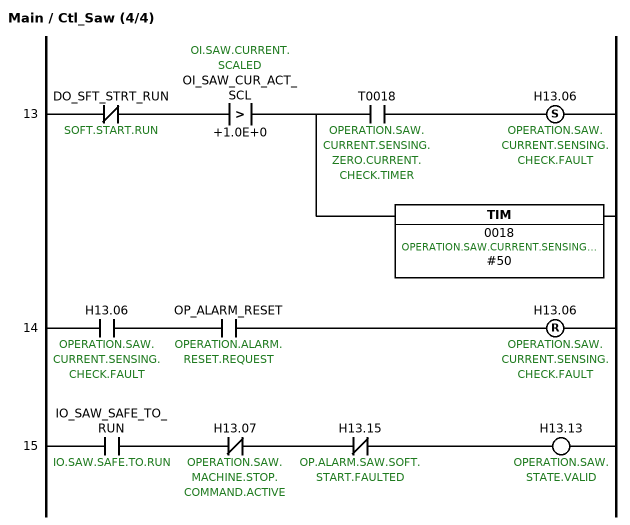
; [picture p72: Main / Ctl_Saw, rungs 13-15]
; rung 13
LDNOT DO_SFT_STRT_RUN  ; SOFT.START.RUN
AND>F(333) OI_SAW_CUR_ACT_SCL +1.0E+0  ; OI.SAW.CURRENT.SCALED
OUT TR0
AND T0018  ; OPERATION.SAW.CURRENT.SENSING.ZERO.CURRENT.CHECK.TIMER
SET H13.06  ; OPERATION.SAW.CURRENT.SENSING.CHECK.FAULT
LD TR0
TIM 0018 #50  ; OPERATION.SAW.CURRENT.SENSING.ZERO.CURRENT.CHECK.TIMER
; rung 14
LD H13.06  ; OPERATION.SAW.CURRENT.SENSING.CHECK.FAULT
AND OP_ALARM_RESET  ; OPERATION.ALARM.RESET.REQUEST
RSET H13.06  ; OPERATION.SAW.CURRENT.SENSING.CHECK.FAULT
; rung 15
LD IO_SAW_SAFE_TO_RUN  ; IO.SAW.SAFE.TO.RUN
ANDNOT H13.07  ; OPERATION.SAW.MACHINE.STOP.COMMAND.ACTIVE
ANDNOT H13.15  ; OP.ALARM.SAW.SOFT.START.FAULTED
OUT H13.13  ; OPERATION.SAW.STATE.VALID

### Section Ctl_Water

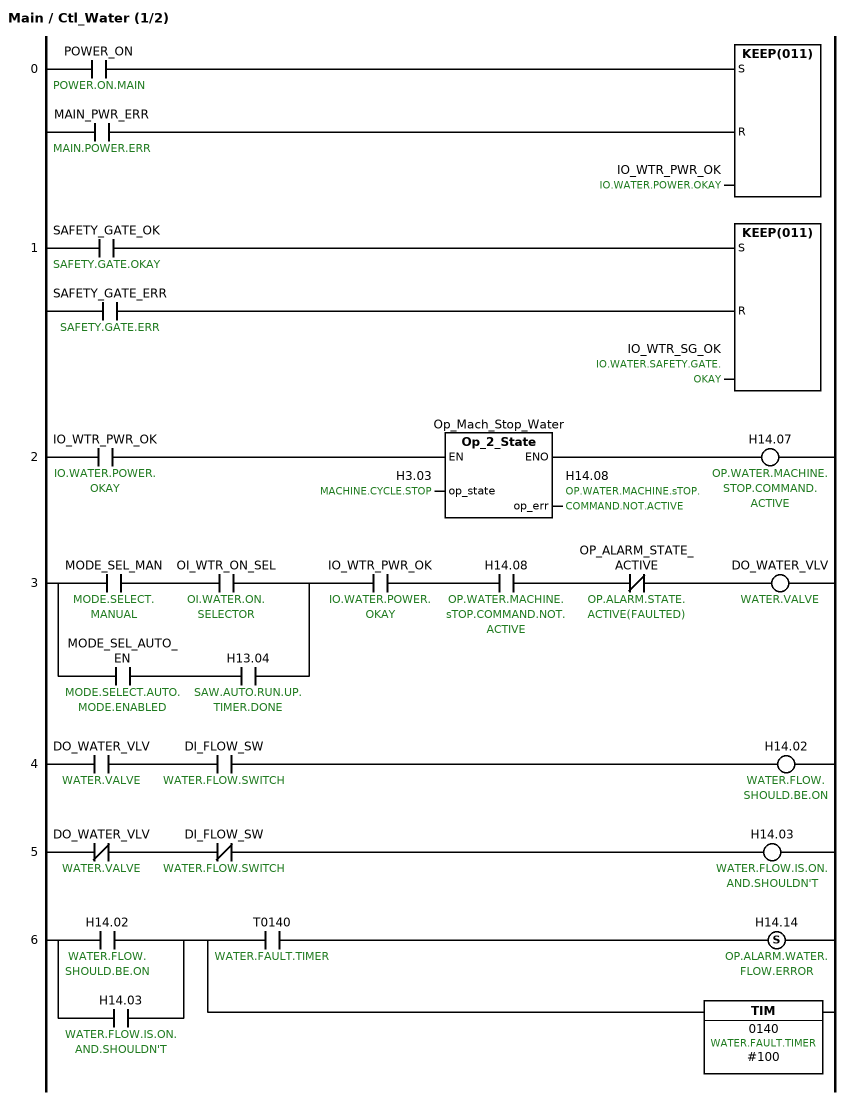
; rung 0
LD POWER_ON  ; POWER.ON.MAIN
LD MAIN_PWR_ERR  ; MAIN.POWER.ERR
KEEP(011) IO_WTR_PWR_OK  ; IO.WATER.POWER.OKAY
; rung 1
LD SAFETY_GATE_OK  ; SAFETY.GATE.OKAY
LD SAFETY_GATE_ERR  ; SAFETY.GATE.ERR
KEEP(011) IO_WTR_SG_OK  ; IO.WATER.SAFETY.GATE.OKAY
; rung 2
LD IO_WTR_PWR_OK  ; IO.WATER.POWER.OKAY
CALL Op_Mach_Stop_Water : Op_2_State (op_state := H3.03, op_err => H14.08)  ; MACHINE.CYCLE.STOP, OP.WATER.MACHINE.sTOP.COMMAND.NOT.ACTIVE
OUT H14.07  ; OP.WATER.MACHINE.STOP.COMMAND.ACTIVE
; rung 3
LD MODE_SEL_MAN  ; MODE.SELECT.MANUAL
AND OI_WTR_ON_SEL  ; OI.WATER.ON.SELECTOR
LD MODE_SEL_AUTO_EN  ; MODE.SELECT.AUTO.MODE.ENABLED
AND H13.04  ; SAW.AUTO.RUN.UP.TIMER.DONE
ORLD
AND IO_WTR_PWR_OK  ; IO.WATER.POWER.OKAY
AND H14.08  ; OP.WATER.MACHINE.sTOP.COMMAND.NOT.ACTIVE
ANDNOT OP_ALARM_STATE_ACTIVE  ; OP.ALARM.STATE.ACTIVE(FAULTED)
OUT DO_WATER_VLV  ; WATER.VALVE
; rung 4
LD DO_WATER_VLV  ; WATER.VALVE
AND DI_FLOW_SW  ; WATER.FLOW.SWITCH
OUT H14.02  ; WATER.FLOW.SHOULD.BE.ON
; rung 5
LDNOT DO_WATER_VLV  ; WATER.VALVE
ANDNOT DI_FLOW_SW  ; WATER.FLOW.SWITCH
OUT H14.03  ; WATER.FLOW.IS.ON.AND.SHOULDN'T
; rung 6
LD H14.02  ; WATER.FLOW.SHOULD.BE.ON
OR H14.03  ; WATER.FLOW.IS.ON.AND.SHOULDN'T
OUT TR0
AND T0140  ; WATER.FAULT.TIMER
SET H14.14  ; OP.ALARM.WATER.FLOW.ERROR
LD TR0
TIM 0140 #100  ; WATER.FAULT.TIMER

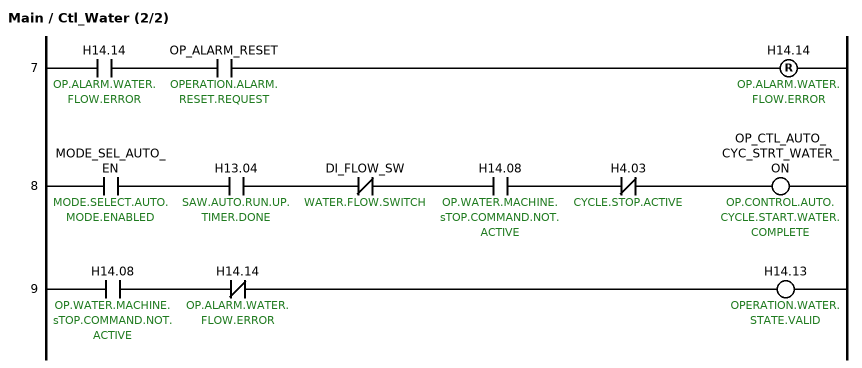
; rung 7
LD H14.14  ; OP.ALARM.WATER.FLOW.ERROR
AND OP_ALARM_RESET  ; OPERATION.ALARM.RESET.REQUEST
RSET H14.14  ; OP.ALARM.WATER.FLOW.ERROR
; rung 8
LD MODE_SEL_AUTO_EN  ; MODE.SELECT.AUTO.MODE.ENABLED
AND H13.04  ; SAW.AUTO.RUN.UP.TIMER.DONE
ANDNOT DI_FLOW_SW  ; WATER.FLOW.SWITCH
AND H14.08  ; OP.WATER.MACHINE.sTOP.COMMAND.NOT.ACTIVE
ANDNOT H4.03  ; CYCLE.STOP.ACTIVE
OUT OP_CTL_AUTO_CYC_STRT_WATER_ON  ; OP.CONTROL.AUTO.CYCLE.START.WATER.COMPLETE
; rung 9
LD H14.08  ; OP.WATER.MACHINE.sTOP.COMMAND.NOT.ACTIVE
ANDNOT H14.14  ; OP.ALARM.WATER.FLOW.ERROR
OUT H14.13  ; OPERATION.WATER.STATE.VALID

### Section Ctl_Lazer

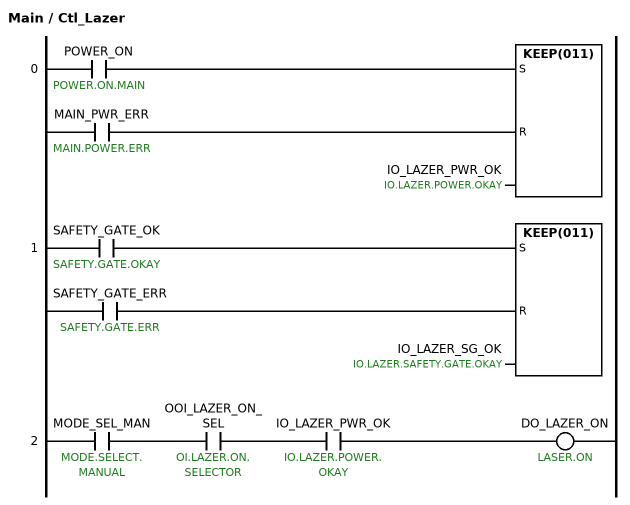
; rung 0
LD POWER_ON  ; POWER.ON.MAIN
LD MAIN_PWR_ERR  ; MAIN.POWER.ERR
KEEP(011) IO_LAZER_PWR_OK  ; IO.LAZER.POWER.OKAY
; rung 1
LD SAFETY_GATE_OK  ; SAFETY.GATE.OKAY
LD SAFETY_GATE_ERR  ; SAFETY.GATE.ERR
KEEP(011) IO_LAZER_SG_OK  ; IO.LAZER.SAFETY.GATE.OKAY
; rung 2
LD MODE_SEL_MAN  ; MODE.SELECT.MANUAL
AND OOI_LAZER_ON_SEL  ; OI.LAZER.ON.SELECTOR
AND IO_LAZER_PWR_OK  ; IO.LAZER.POWER.OKAY
OUT DO_LAZER_ON  ; LASER.ON

### Section Init_Recipe

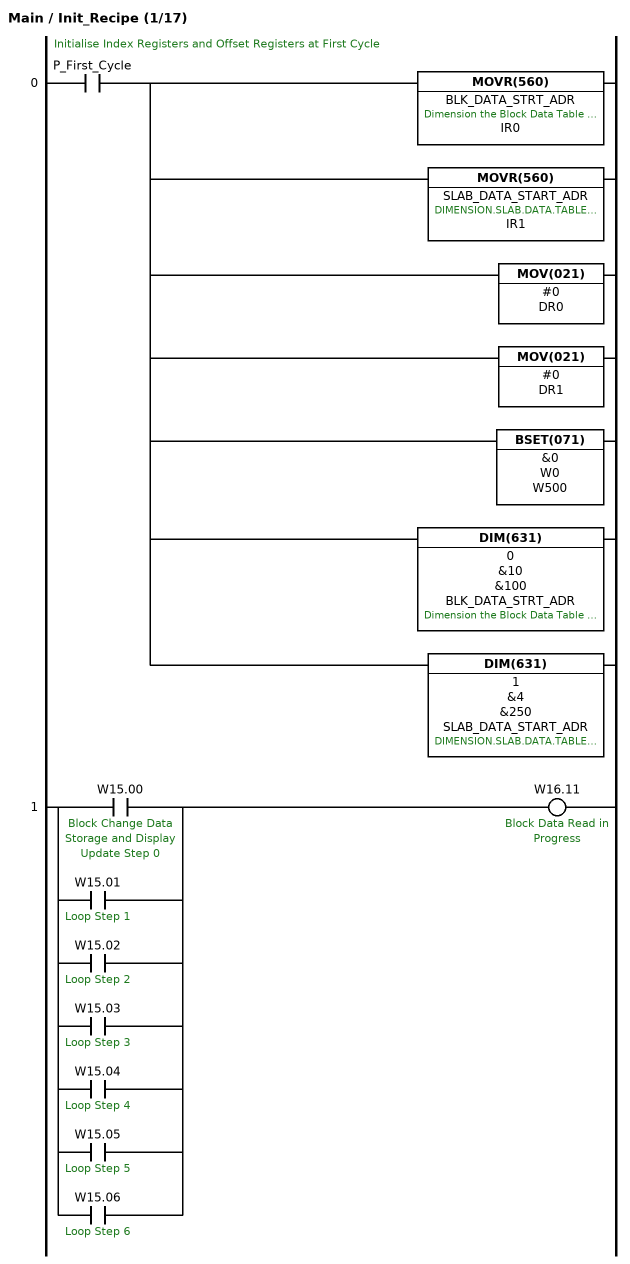
; rung 0: Initialise Index Registers and Offset Registers at First Cycle
LD P_First_Cycle
MOVR(560) BLK_DATA_STRT_ADR IR0  ; Dimension the Block Data Table - Start Address
MOVR(560) SLAB_DATA_START_ADR IR1  ; DIMENSION.SLAB.DATA.TABLE.START.ADDRESS
MOV(021) #0 DR0
MOV(021) #0 DR1
BSET(071) &0 W0 W500
DIM(631) 0 &10 &100 BLK_DATA_STRT_ADR  ; Dimension the Block Data Table - Start Address
DIM(631) 1 &4 &250 SLAB_DATA_START_ADR  ; DIMENSION.SLAB.DATA.TABLE.START.ADDRESS
; rung 1
LD W15.00  ; Block Change Data Storage and Display Update Step 0
OR W15.01  ; Loop Step 1
OR W15.02  ; Loop Step 2
OR W15.03  ; Loop Step 3
OR W15.04  ; Loop Step 4
OR W15.05  ; Loop Step 5
OR W15.06  ; Loop Step 6
OUT W16.11  ; Block Data Read in Progress

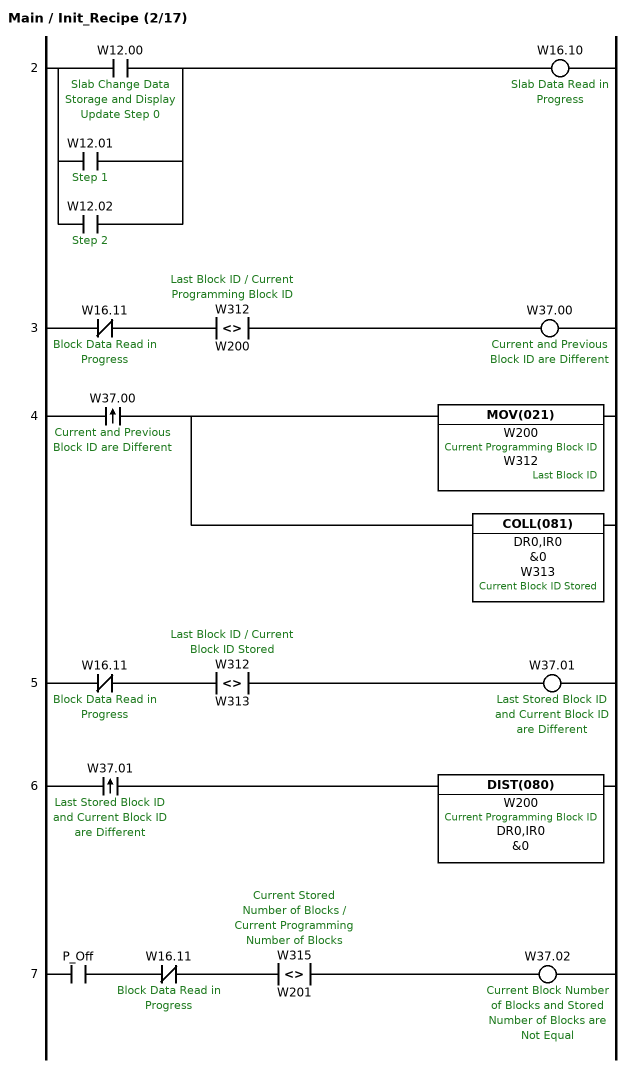
; rung 2
LD W12.00  ; Slab Change Data Storage and Display Update Step 0
OR W12.01  ; Step 1
OR W12.02  ; Step 2
OUT W16.10  ; Slab Data Read in Progress
; rung 3
LDNOT W16.11  ; Block Data Read in Progress
AND<>(305) W312 W200  ; Last Block ID, Current Programming Block ID
OUT W37.00  ; Current and Previous Block ID are Different
; rung 4
@LD W37.00  ; Current and Previous Block ID are Different
MOV(021) W200 W312  ; Current Programming Block ID, Last Block ID
COLL(081) DR0,IR0 &0 W313  ; Current Block ID Stored
; rung 5
LDNOT W16.11  ; Block Data Read in Progress
AND<>(305) W312 W313  ; Last Block ID, Current Block ID Stored
OUT W37.01  ; Last Stored Block ID and Current Block ID are Different
; rung 6
@LD W37.01  ; Last Stored Block ID and Current Block ID are Different
DIST(080) W200 DR0,IR0 &0  ; Current Programming Block ID
; rung 7
LD P_Off
ANDNOT W16.11  ; Block Data Read in Progress
AND<>(305) W315 W201  ; Current Stored Number of Blocks, Current Programming Number of Blocks
OUT W37.02  ; Current Block Number of Blocks and Stored Number of Blocks are Not Equal

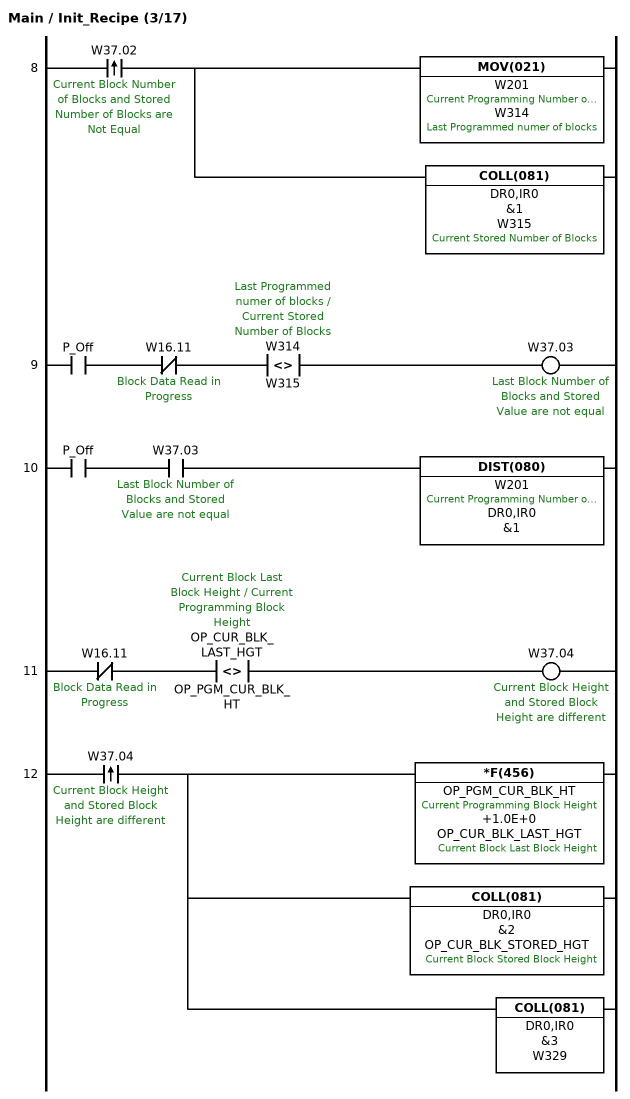
; rung 8
@LD W37.02  ; Current Block Number of Blocks and Stored Number of Blocks are Not Equal
MOV(021) W201 W314  ; Current Programming Number of Blocks, Last Programmed numer of blocks
COLL(081) DR0,IR0 &1 W315  ; Current Stored Number of Blocks
; rung 9
LD P_Off
ANDNOT W16.11  ; Block Data Read in Progress
AND<>(305) W314 W315  ; Last Programmed numer of blocks, Current Stored Number of Blocks
OUT W37.03  ; Last Block Number of Blocks and Stored Value are not equal
; rung 10
LD P_Off
AND W37.03  ; Last Block Number of Blocks and Stored Value are not equal
DIST(080) W201 DR0,IR0 &1  ; Current Programming Number of Blocks
; rung 11
LDNOT W16.11  ; Block Data Read in Progress
AND<>F(330) OP_CUR_BLK_LAST_HGT OP_PGM_CUR_BLK_HT  ; Current Block Last Block Height, Current Programming Block Height
OUT W37.04  ; Current Block Height and Stored Block Height are different
; rung 12
@LD W37.04  ; Current Block Height and Stored Block Height are different
*F(456) OP_PGM_CUR_BLK_HT +1.0E+0 OP_CUR_BLK_LAST_HGT  ; Current Programming Block Height, Current Block Last Block Height
COLL(081) DR0,IR0 &2 OP_CUR_BLK_STORED_HGT  ; Current Block Stored Block Height
COLL(081) DR0,IR0 &3 W329

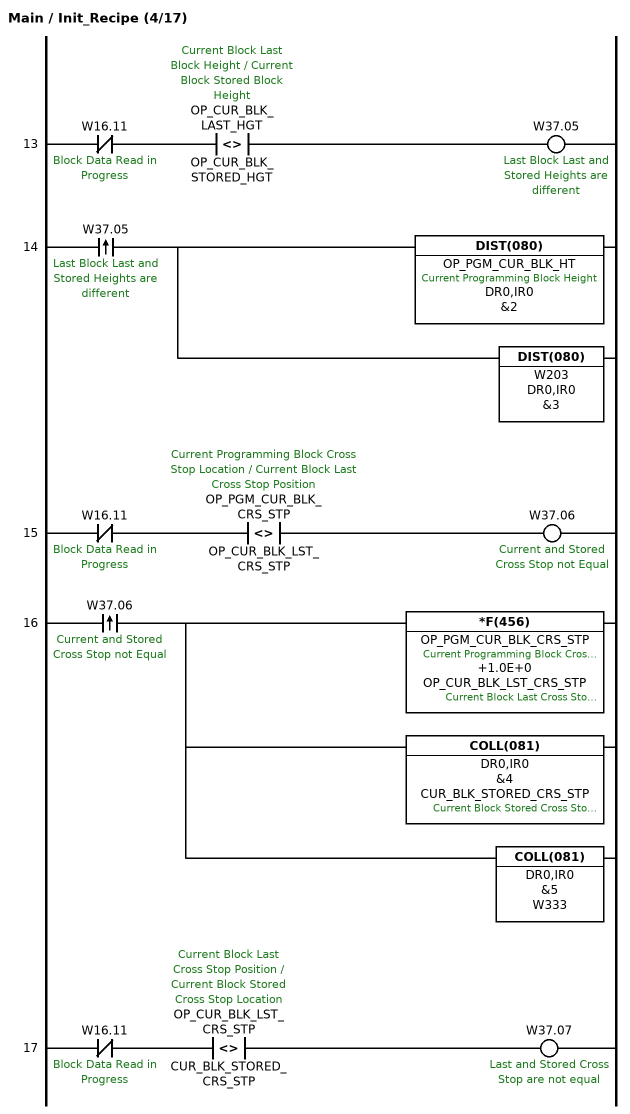
; rung 13
LDNOT W16.11  ; Block Data Read in Progress
AND<>F(330) OP_CUR_BLK_LAST_HGT OP_CUR_BLK_STORED_HGT  ; Current Block Last Block Height, Current Block Stored Block Height
OUT W37.05  ; Last Block Last and Stored Heights are different
; rung 14
@LD W37.05  ; Last Block Last and Stored Heights are different
DIST(080) OP_PGM_CUR_BLK_HT DR0,IR0 &2  ; Current Programming Block Height
DIST(080) W203 DR0,IR0 &3
; rung 15
LDNOT W16.11  ; Block Data Read in Progress
AND<>F(330) OP_PGM_CUR_BLK_CRS_STP OP_CUR_BLK_LST_CRS_STP  ; Current Programming Block Cross Stop Location, Current Block Last Cross Stop Position
OUT W37.06  ; Current and Stored Cross Stop not Equal
; rung 16
@LD W37.06  ; Current and Stored Cross Stop not Equal
*F(456) OP_PGM_CUR_BLK_CRS_STP +1.0E+0 OP_CUR_BLK_LST_CRS_STP  ; Current Programming Block Cross Stop Location, Current Block Last Cross Stop Position
COLL(081) DR0,IR0 &4 CUR_BLK_STORED_CRS_STP  ; Current Block Stored Cross Stop Location
COLL(081) DR0,IR0 &5 W333
; rung 17
LDNOT W16.11  ; Block Data Read in Progress
AND<>F(330) OP_CUR_BLK_LST_CRS_STP CUR_BLK_STORED_CRS_STP  ; Current Block Last Cross Stop Position, Current Block Stored Cross Stop Location
OUT W37.07  ; Last and Stored Cross Stop are not equal

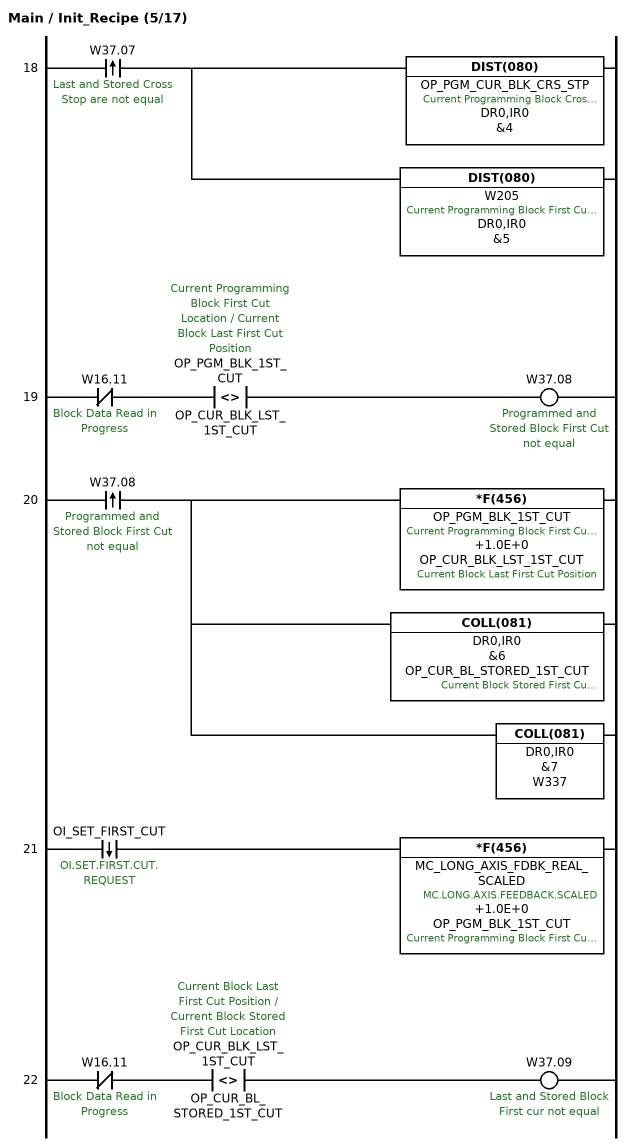
; rung 18
@LD W37.07  ; Last and Stored Cross Stop are not equal
DIST(080) OP_PGM_CUR_BLK_CRS_STP DR0,IR0 &4  ; Current Programming Block Cross Stop Location
DIST(080) W205 DR0,IR0 &5  ; Current Programming Block First Cut Location
; rung 19
LDNOT W16.11  ; Block Data Read in Progress
AND<>F(330) OP_PGM_BLK_1ST_CUT OP_CUR_BLK_LST_1ST_CUT  ; Current Programming Block First Cut Location, Current Block Last First Cut Position
OUT W37.08  ; Programmed and Stored Block First Cut not equal
; rung 20
@LD W37.08  ; Programmed and Stored Block First Cut not equal
*F(456) OP_PGM_BLK_1ST_CUT +1.0E+0 OP_CUR_BLK_LST_1ST_CUT  ; Current Programming Block First Cut Location, Current Block Last First Cut Position
COLL(081) DR0,IR0 &6 OP_CUR_BL_STORED_1ST_CUT  ; Current Block Stored First Cut Location
COLL(081) DR0,IR0 &7 W337
; rung 21
%LD OI_SET_FIRST_CUT  ; OI.SET.FIRST.CUT.REQUEST
*F(456) MC_LONG_AXIS_FDBK_REAL_SCALED +1.0E+0 OP_PGM_BLK_1ST_CUT  ; MC.LONG.AXIS.FEEDBACK.SCALED, Current Programming Block First Cut Location
; rung 22
LDNOT W16.11  ; Block Data Read in Progress
AND<>F(330) OP_CUR_BLK_LST_1ST_CUT OP_CUR_BL_STORED_1ST_CUT  ; Current Block Last First Cut Position, Current Block Stored First Cut Location
OUT W37.09  ; Last and Stored Block First cur not equal

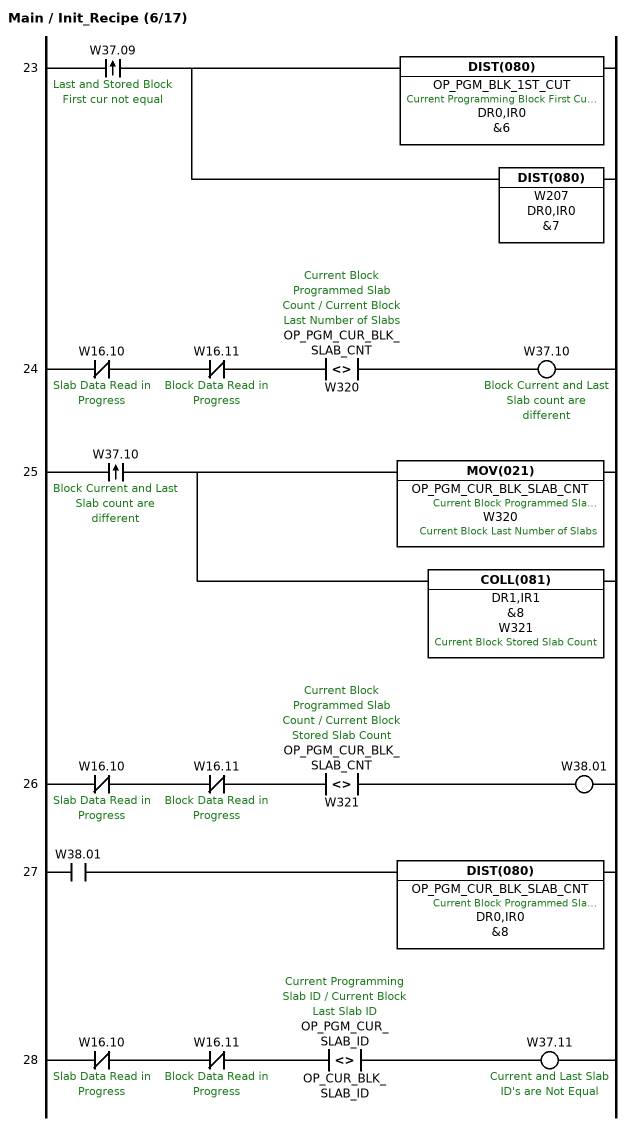
; rung 23
@LD W37.09  ; Last and Stored Block First cur not equal
DIST(080) OP_PGM_BLK_1ST_CUT DR0,IR0 &6  ; Current Programming Block First Cut Location
DIST(080) W207 DR0,IR0 &7
; rung 24
LDNOT W16.10  ; Slab Data Read in Progress
ANDNOT W16.11  ; Block Data Read in Progress
AND<>(305) OP_PGM_CUR_BLK_SLAB_CNT W320  ; Current Block Programmed Slab Count, Current Block Last Number of Slabs
OUT W37.10  ; Block Current and Last Slab count are different
; rung 25
@LD W37.10  ; Block Current and Last Slab count are different
MOV(021) OP_PGM_CUR_BLK_SLAB_CNT W320  ; Current Block Programmed Slab Count, Current Block Last Number of Slabs
COLL(081) DR1,IR1 &8 W321  ; Current Block Stored Slab Count
; rung 26
LDNOT W16.10  ; Slab Data Read in Progress
ANDNOT W16.11  ; Block Data Read in Progress
AND<>(305) OP_PGM_CUR_BLK_SLAB_CNT W321  ; Current Block Programmed Slab Count, Current Block Stored Slab Count
OUT W38.01
; rung 27
LD W38.01
DIST(080) OP_PGM_CUR_BLK_SLAB_CNT DR0,IR0 &8  ; Current Block Programmed Slab Count
; rung 28
LDNOT W16.10  ; Slab Data Read in Progress
ANDNOT W16.11  ; Block Data Read in Progress
AND<>(305) OP_PGM_CUR_SLAB_ID OP_CUR_BLK_SLAB_ID  ; Current Programming Slab ID, Current Block Last Slab ID
OUT W37.11  ; Current and Last Slab ID's are Not Equal

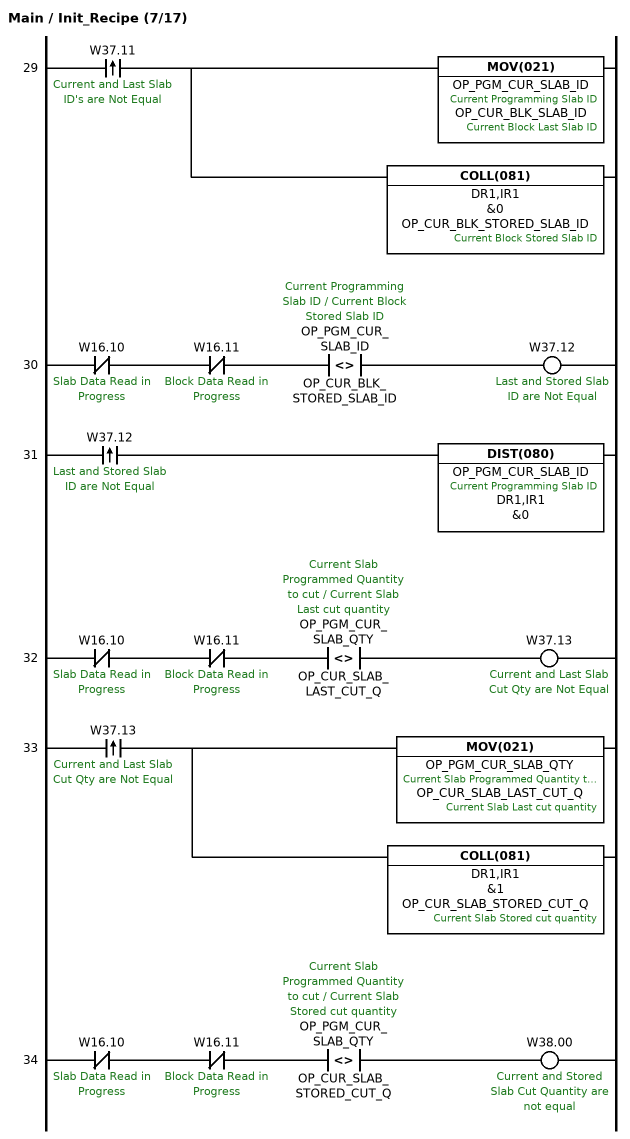
; rung 29
@LD W37.11  ; Current and Last Slab ID's are Not Equal
MOV(021) OP_PGM_CUR_SLAB_ID OP_CUR_BLK_SLAB_ID  ; Current Programming Slab ID, Current Block Last Slab ID
COLL(081) DR1,IR1 &0 OP_CUR_BLK_STORED_SLAB_ID  ; Current Block Stored Slab ID
; rung 30
LDNOT W16.10  ; Slab Data Read in Progress
ANDNOT W16.11  ; Block Data Read in Progress
AND<>(305) OP_PGM_CUR_SLAB_ID OP_CUR_BLK_STORED_SLAB_ID  ; Current Programming Slab ID, Current Block Stored Slab ID
OUT W37.12  ; Last and Stored Slab ID are Not Equal
; rung 31
@LD W37.12  ; Last and Stored Slab ID are Not Equal
DIST(080) OP_PGM_CUR_SLAB_ID DR1,IR1 &0  ; Current Programming Slab ID
; rung 32
LDNOT W16.10  ; Slab Data Read in Progress
ANDNOT W16.11  ; Block Data Read in Progress
AND<>(305) OP_PGM_CUR_SLAB_QTY OP_CUR_SLAB_LAST_CUT_Q  ; Current Slab Programmed Quantity to cut, Current Slab Last cut quantity
OUT W37.13  ; Current and Last Slab Cut Qty are Not Equal
; rung 33
@LD W37.13  ; Current and Last Slab Cut Qty are Not Equal
MOV(021) OP_PGM_CUR_SLAB_QTY OP_CUR_SLAB_LAST_CUT_Q  ; Current Slab Programmed Quantity to cut, Current Slab Last cut quantity
COLL(081) DR1,IR1 &1 OP_CUR_SLAB_STORED_CUT_Q  ; Current Slab Stored cut quantity
; rung 34
LDNOT W16.10  ; Slab Data Read in Progress
ANDNOT W16.11  ; Block Data Read in Progress
AND<>(305) OP_PGM_CUR_SLAB_QTY OP_CUR_SLAB_STORED_CUT_Q  ; Current Slab Programmed Quantity to cut, Current Slab Stored cut quantity
OUT W38.00  ; Current and Stored Slab Cut Quantity are not equal

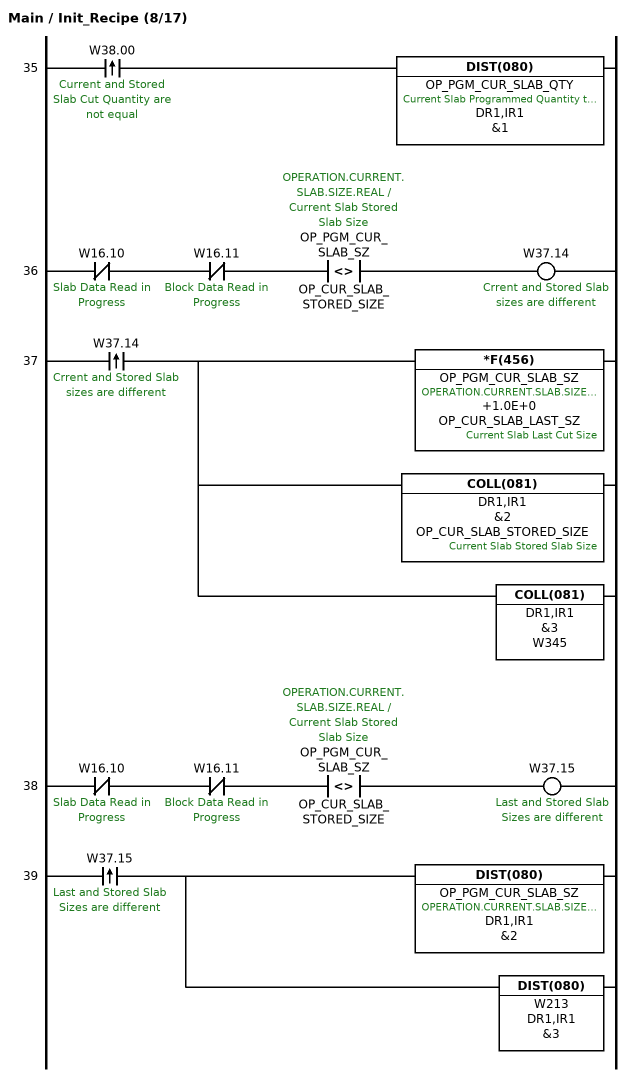
; rung 35
@LD W38.00  ; Current and Stored Slab Cut Quantity are not equal
DIST(080) OP_PGM_CUR_SLAB_QTY DR1,IR1 &1  ; Current Slab Programmed Quantity to cut
; rung 36
LDNOT W16.10  ; Slab Data Read in Progress
ANDNOT W16.11  ; Block Data Read in Progress
AND<>F(330) OP_PGM_CUR_SLAB_SZ OP_CUR_SLAB_STORED_SIZE  ; OPERATION.CURRENT.SLAB.SIZE.REAL, Current Slab Stored Slab Size
OUT W37.14  ; Crrent and Stored Slab sizes are different
; rung 37
@LD W37.14  ; Crrent and Stored Slab sizes are different
*F(456) OP_PGM_CUR_SLAB_SZ +1.0E+0 OP_CUR_SLAB_LAST_SZ  ; OPERATION.CURRENT.SLAB.SIZE.REAL, Current Slab Last Cut Size
COLL(081) DR1,IR1 &2 OP_CUR_SLAB_STORED_SIZE  ; Current Slab Stored Slab Size
COLL(081) DR1,IR1 &3 W345
; rung 38
LDNOT W16.10  ; Slab Data Read in Progress
ANDNOT W16.11  ; Block Data Read in Progress
AND<>F(330) OP_PGM_CUR_SLAB_SZ OP_CUR_SLAB_STORED_SIZE  ; OPERATION.CURRENT.SLAB.SIZE.REAL, Current Slab Stored Slab Size
OUT W37.15  ; Last and Stored Slab Sizes are different
; rung 39
@LD W37.15  ; Last and Stored Slab Sizes are different
DIST(080) OP_PGM_CUR_SLAB_SZ DR1,IR1 &2  ; OPERATION.CURRENT.SLAB.SIZE.REAL
DIST(080) W213 DR1,IR1 &3

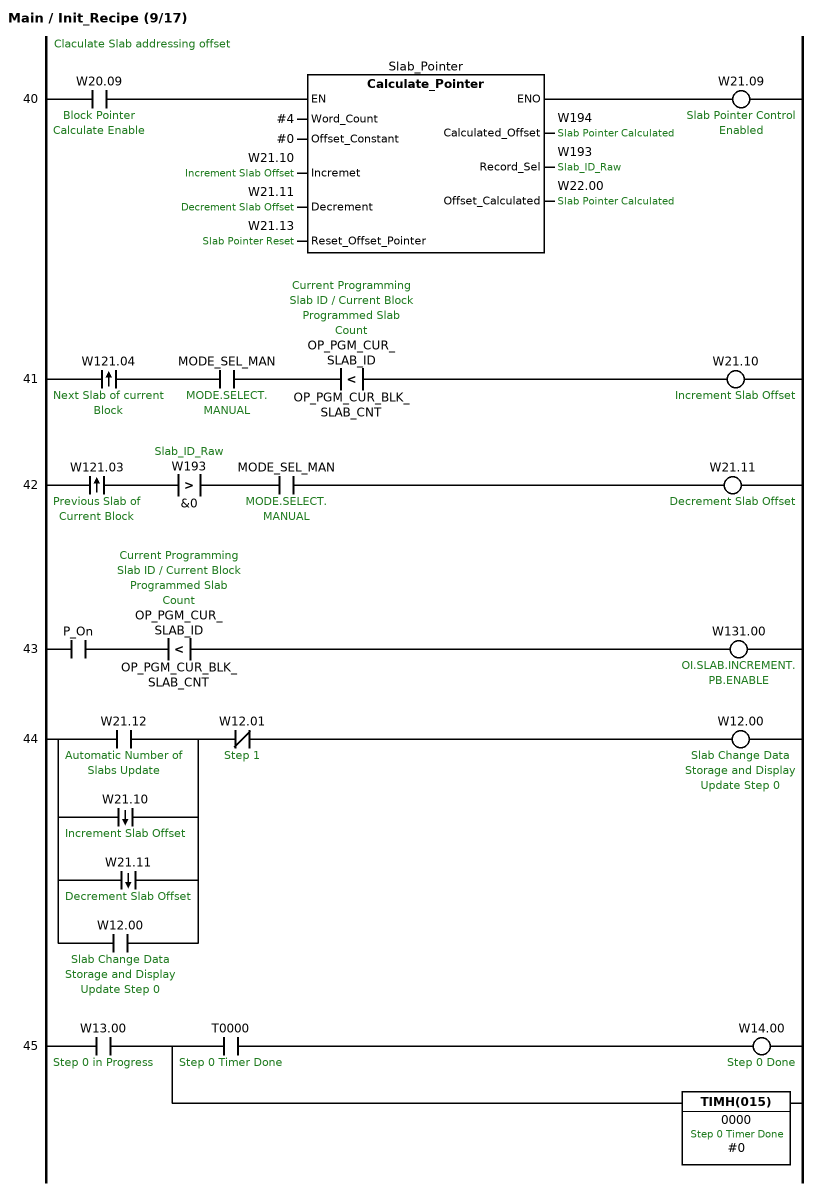
; rung 40: Claculate Slab addressing offset
LD W20.09  ; Block Pointer Calculate Enable
CALL Slab_Pointer : Calculate_Pointer (Word_Count := #4, Offset_Constant := #0, Incremet := W21.10, Decrement := W21.11, Reset_Offset_Pointer := W21.13, Calculated_Offset => W194, Record_Sel => W193, Offset_Calculated => W22.00)  ; Increment Slab Offset, Decrement Slab Offset, Slab Pointer Reset, Slab Pointer Calculated, Slab_ID_Raw
OUT W21.09  ; Slab Pointer Control Enabled
; rung 41
@LD W121.04  ; Next Slab of current Block
AND MODE_SEL_MAN  ; MODE.SELECT.MANUAL
AND<(310) OP_PGM_CUR_SLAB_ID OP_PGM_CUR_BLK_SLAB_CNT  ; Current Programming Slab ID, Current Block Programmed Slab Count
OUT W21.10  ; Increment Slab Offset
; rung 42
@LD W121.03  ; Previous Slab of Current Block
AND>(320) W193 &0  ; Slab_ID_Raw
AND MODE_SEL_MAN  ; MODE.SELECT.MANUAL
OUT W21.11  ; Decrement Slab Offset
; rung 43
LD P_On
AND<(310) OP_PGM_CUR_SLAB_ID OP_PGM_CUR_BLK_SLAB_CNT  ; Current Programming Slab ID, Current Block Programmed Slab Count
OUT W131.00  ; OI.SLAB.INCREMENT.PB.ENABLE
; rung 44
LD W21.12  ; Automatic Number of Slabs Update
%OR W21.10  ; Increment Slab Offset
%OR W21.11  ; Decrement Slab Offset
OR W12.00  ; Slab Change Data Storage and Display Update Step 0
ANDNOT W12.01  ; Step 1
OUT W12.00  ; Slab Change Data Storage and Display Update Step 0
; rung 45
LD W13.00  ; Step 0 in Progress
OUT TR0
AND T0000  ; Step 0 Timer Done
OUT W14.00  ; Step 0 Done
LD TR0
TIMH(015) 0000 #0  ; Step 0 Timer Done

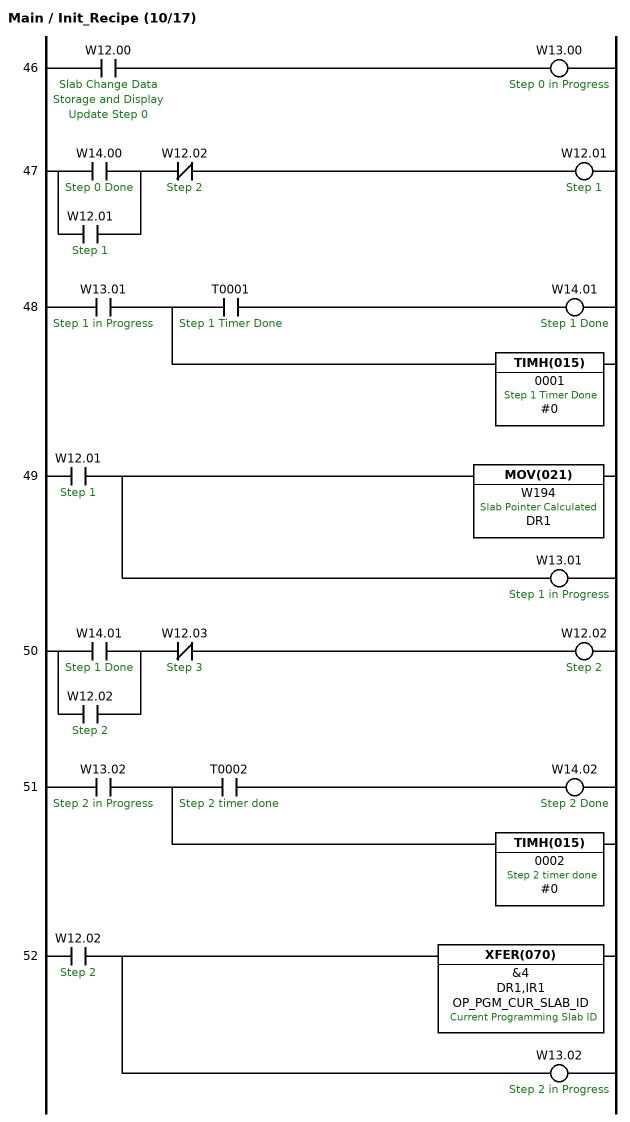
; rung 46
LD W12.00  ; Slab Change Data Storage and Display Update Step 0
OUT W13.00  ; Step 0 in Progress
; rung 47
LD W14.00  ; Step 0 Done
OR W12.01  ; Step 1
ANDNOT W12.02  ; Step 2
OUT W12.01  ; Step 1
; rung 48
LD W13.01  ; Step 1 in Progress
OUT TR0
AND T0001  ; Step 1 Timer Done
OUT W14.01  ; Step 1 Done
LD TR0
TIMH(015) 0001 #0  ; Step 1 Timer Done
; rung 49
LD W12.01  ; Step 1
MOV(021) W194 DR1  ; Slab Pointer Calculated
OUT W13.01  ; Step 1 in Progress
; rung 50
LD W14.01  ; Step 1 Done
OR W12.02  ; Step 2
ANDNOT W12.03  ; Step 3
OUT W12.02  ; Step 2
; rung 51
LD W13.02  ; Step 2 in Progress
OUT TR0
AND T0002  ; Step 2 timer done
OUT W14.02  ; Step 2 Done
LD TR0
TIMH(015) 0002 #0  ; Step 2 timer done
; rung 52
LD W12.02  ; Step 2
XFER(070) &4 DR1,IR1 OP_PGM_CUR_SLAB_ID  ; Current Programming Slab ID
OUT W13.02  ; Step 2 in Progress

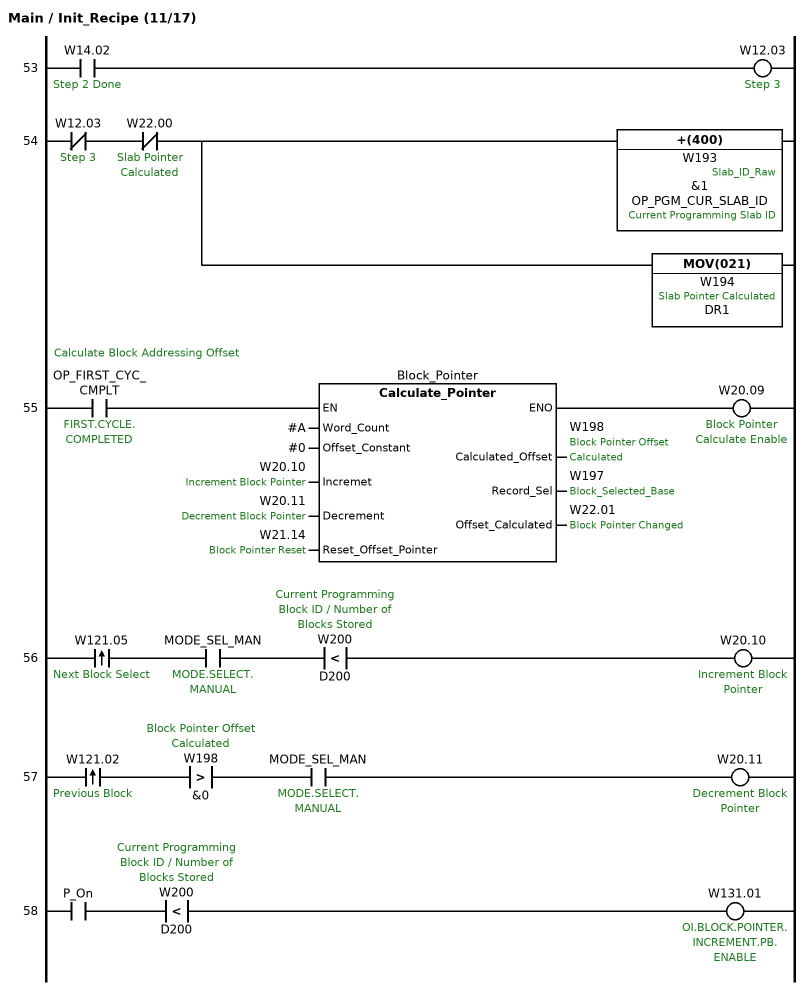
; rung 53
LD W14.02  ; Step 2 Done
OUT W12.03  ; Step 3
; rung 54
LDNOT W12.03  ; Step 3
ANDNOT W22.00  ; Slab Pointer Calculated
+(400) W193 &1 OP_PGM_CUR_SLAB_ID  ; Slab_ID_Raw, Current Programming Slab ID
MOV(021) W194 DR1  ; Slab Pointer Calculated
; rung 55: Calculate Block Addressing Offset
LD OP_FIRST_CYC_CMPLT  ; FIRST.CYCLE.COMPLETED
CALL Block_Pointer : Calculate_Pointer (Word_Count := #A, Offset_Constant := #0, Incremet := W20.10, Decrement := W20.11, Reset_Offset_Pointer := W21.14, Calculated_Offset => W198, Record_Sel => W197, Offset_Calculated => W22.01)  ; Increment Block Pointer, Decrement Block Pointer, Block Pointer Reset, Block Pointer Offset Calculated, Block_Selected_Base, Block Pointer Changed
OUT W20.09  ; Block Pointer Calculate Enable
; rung 56
@LD W121.05  ; Next Block Select
AND MODE_SEL_MAN  ; MODE.SELECT.MANUAL
AND<(310) W200 D200  ; Current Programming Block ID, Number of Blocks Stored
OUT W20.10  ; Increment Block Pointer
; rung 57
@LD W121.02  ; Previous Block
AND>(320) W198 &0  ; Block Pointer Offset Calculated
AND MODE_SEL_MAN  ; MODE.SELECT.MANUAL
OUT W20.11  ; Decrement Block Pointer
; rung 58
LD P_On
AND<(310) W200 D200  ; Current Programming Block ID, Number of Blocks Stored
OUT W131.01  ; OI.BLOCK.POINTER.INCREMENT.PB.ENABLE

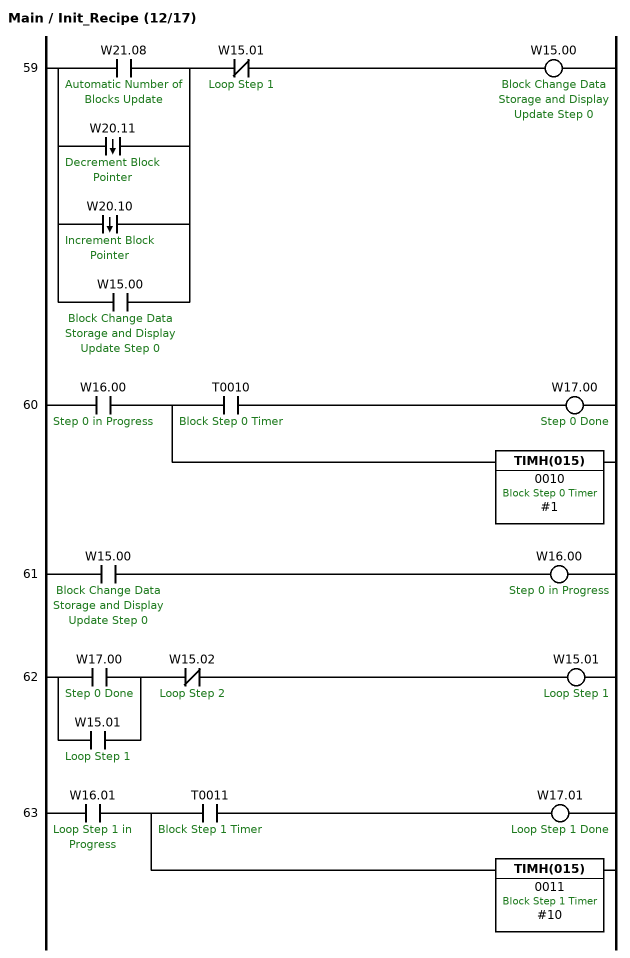
; rung 59
LD W21.08  ; Automatic Number of Blocks Update
%OR W20.11  ; Decrement Block Pointer
%OR W20.10  ; Increment Block Pointer
OR W15.00  ; Block Change Data Storage and Display Update Step 0
ANDNOT W15.01  ; Loop Step 1
OUT W15.00  ; Block Change Data Storage and Display Update Step 0
; rung 60
LD W16.00  ; Step 0 in Progress
OUT TR0
AND T0010  ; Block Step 0 Timer
OUT W17.00  ; Step 0 Done
LD TR0
TIMH(015) 0010 #1  ; Block Step 0 Timer
; rung 61
LD W15.00  ; Block Change Data Storage and Display Update Step 0
OUT W16.00  ; Step 0 in Progress
; rung 62
LD W17.00  ; Step 0 Done
OR W15.01  ; Loop Step 1
ANDNOT W15.02  ; Loop Step 2
OUT W15.01  ; Loop Step 1
; rung 63
LD W16.01  ; Loop Step 1 in Progress
OUT TR0
AND T0011  ; Block Step 1 Timer
OUT W17.01  ; Loop Step 1 Done
LD TR0
TIMH(015) 0011 #10  ; Block Step 1 Timer

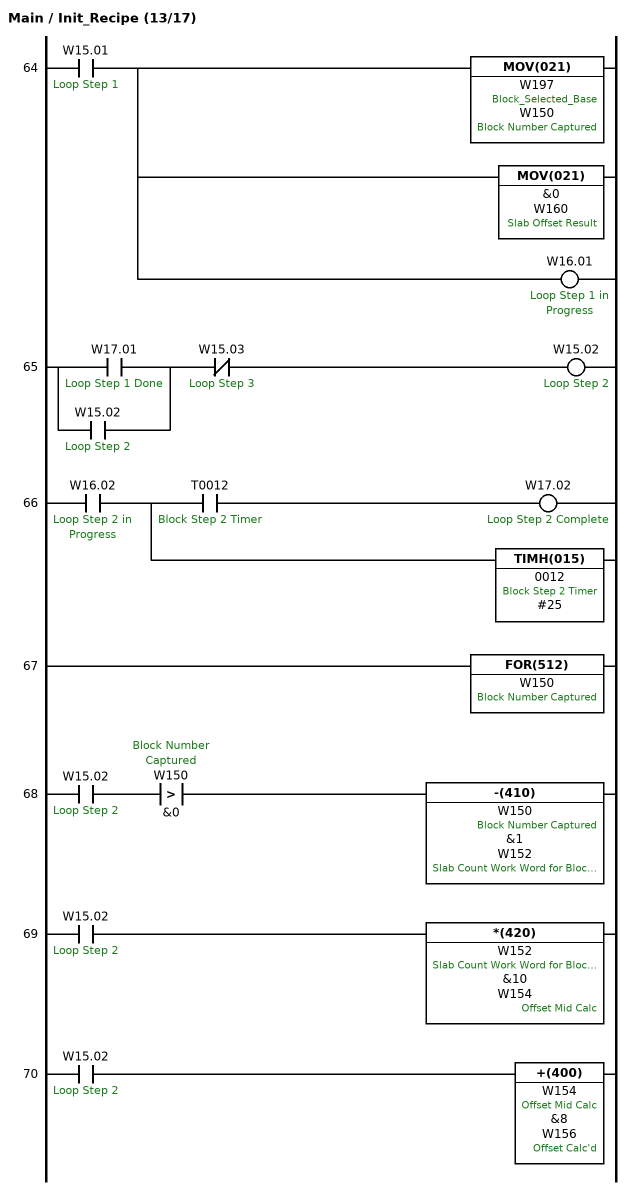
; rung 64
LD W15.01  ; Loop Step 1
MOV(021) W197 W150  ; Block_Selected_Base, Block Number Captured
MOV(021) &0 W160  ; Slab Offset Result
OUT W16.01  ; Loop Step 1 in Progress
; rung 65
LD W17.01  ; Loop Step 1 Done
OR W15.02  ; Loop Step 2
ANDNOT W15.03  ; Loop Step 3
OUT W15.02  ; Loop Step 2
; rung 66
LD W16.02  ; Loop Step 2 in Progress
OUT TR0
AND T0012  ; Block Step 2 Timer
OUT W17.02  ; Loop Step 2 Complete
LD TR0
TIMH(015) 0012 #25  ; Block Step 2 Timer
; rung 67
FOR(512) W150  ; Block Number Captured
; rung 68
LD W15.02  ; Loop Step 2
AND>(320) W150 &0  ; Block Number Captured
-(410) W150 &1 W152  ; Block Number Captured, Slab Count Work Word for Block Pointer
; rung 69
LD W15.02  ; Loop Step 2
*(420) W152 &10 W154  ; Slab Count Work Word for Block Pointer, Offset Mid Calc
; rung 70
LD W15.02  ; Loop Step 2
+(400) W154 &8 W156  ; Offset Mid Calc, Offset Calc'd

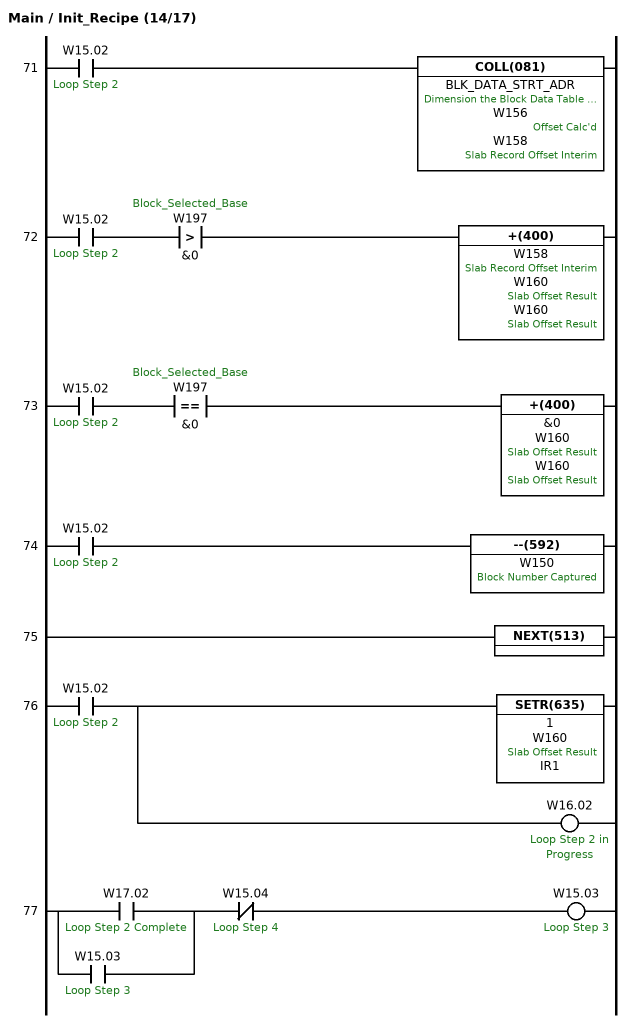
; rung 71
LD W15.02  ; Loop Step 2
COLL(081) BLK_DATA_STRT_ADR W156 W158  ; Dimension the Block Data Table - Start Address, Offset Calc'd, Slab Record Offset Interim
; rung 72
LD W15.02  ; Loop Step 2
AND>(320) W197 &0  ; Block_Selected_Base
+(400) W158 W160 W160  ; Slab Record Offset Interim, Slab Offset Result
; rung 73
LD W15.02  ; Loop Step 2
AND=(300) W197 &0  ; Block_Selected_Base
+(400) &0 W160 W160  ; Slab Offset Result
; rung 74
LD W15.02  ; Loop Step 2
--(592) W150  ; Block Number Captured
; rung 75
NEXT(513)
; rung 76
LD W15.02  ; Loop Step 2
SETR(635) 1 W160 IR1  ; Slab Offset Result
OUT W16.02  ; Loop Step 2 in Progress
; rung 77
LD W17.02  ; Loop Step 2 Complete
OR W15.03  ; Loop Step 3
ANDNOT W15.04  ; Loop Step 4
OUT W15.03  ; Loop Step 3

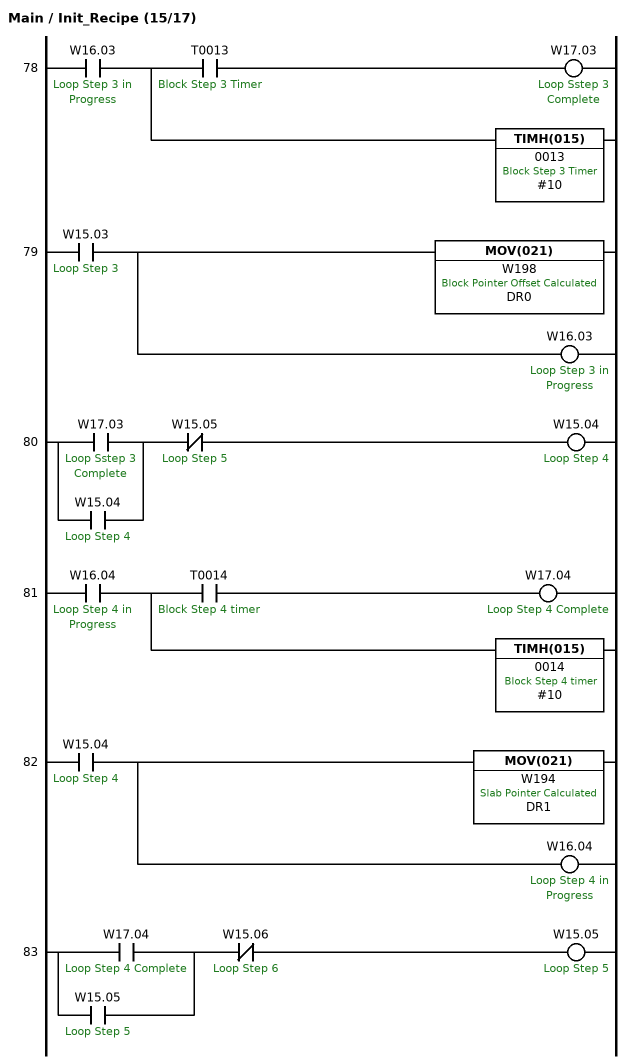
; rung 78
LD W16.03  ; Loop Step 3 in Progress
OUT TR0
AND T0013  ; Block Step 3 Timer
OUT W17.03  ; Loop Sstep 3 Complete
LD TR0
TIMH(015) 0013 #10  ; Block Step 3 Timer
; rung 79
LD W15.03  ; Loop Step 3
MOV(021) W198 DR0  ; Block Pointer Offset Calculated
OUT W16.03  ; Loop Step 3 in Progress
; rung 80
LD W17.03  ; Loop Sstep 3 Complete
OR W15.04  ; Loop Step 4
ANDNOT W15.05  ; Loop Step 5
OUT W15.04  ; Loop Step 4
; rung 81
LD W16.04  ; Loop Step 4 in Progress
OUT TR0
AND T0014  ; Block Step 4 timer
OUT W17.04  ; Loop Step 4 Complete
LD TR0
TIMH(015) 0014 #10  ; Block Step 4 timer
; rung 82
LD W15.04  ; Loop Step 4
MOV(021) W194 DR1  ; Slab Pointer Calculated
OUT W16.04  ; Loop Step 4 in Progress
; rung 83
LD W17.04  ; Loop Step 4 Complete
OR W15.05  ; Loop Step 5
ANDNOT W15.06  ; Loop Step 6
OUT W15.05  ; Loop Step 5

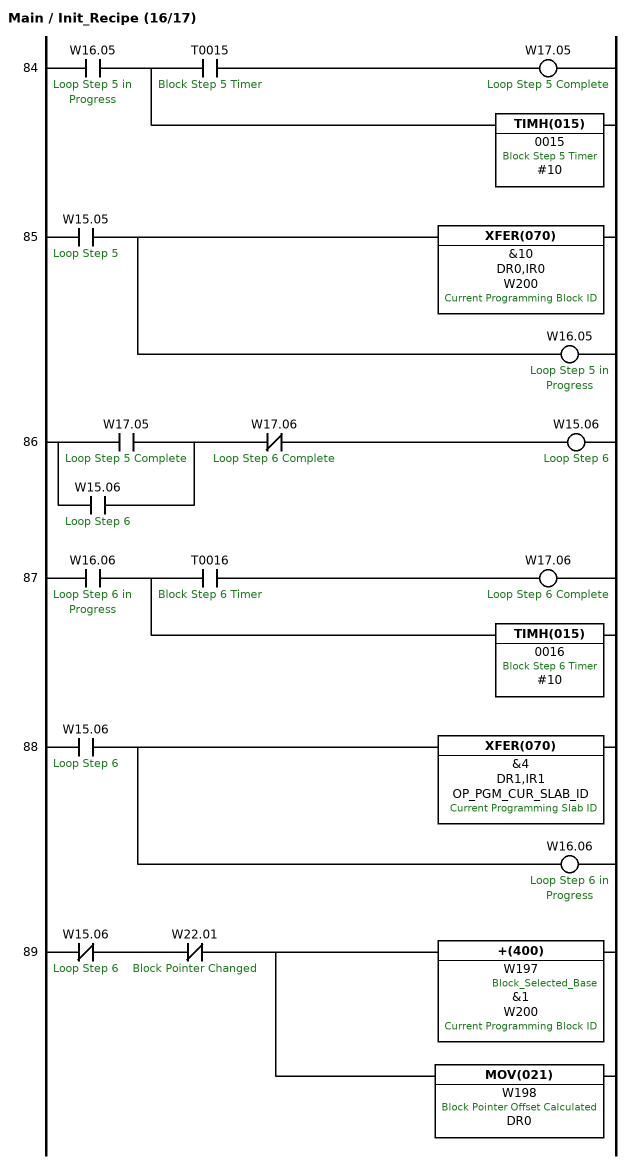
; rung 84
LD W16.05  ; Loop Step 5 in Progress
OUT TR0
AND T0015  ; Block Step 5 Timer
OUT W17.05  ; Loop Step 5 Complete
LD TR0
TIMH(015) 0015 #10  ; Block Step 5 Timer
; rung 85
LD W15.05  ; Loop Step 5
XFER(070) &10 DR0,IR0 W200  ; Current Programming Block ID
OUT W16.05  ; Loop Step 5 in Progress
; rung 86
LD W17.05  ; Loop Step 5 Complete
OR W15.06  ; Loop Step 6
ANDNOT W17.06  ; Loop Step 6 Complete
OUT W15.06  ; Loop Step 6
; rung 87
LD W16.06  ; Loop Step 6 in Progress
OUT TR0
AND T0016  ; Block Step 6 Timer
OUT W17.06  ; Loop Step 6 Complete
LD TR0
TIMH(015) 0016 #10  ; Block Step 6 Timer
; rung 88
LD W15.06  ; Loop Step 6
XFER(070) &4 DR1,IR1 OP_PGM_CUR_SLAB_ID  ; Current Programming Slab ID
OUT W16.06  ; Loop Step 6 in Progress
; rung 89
LDNOT W15.06  ; Loop Step 6
ANDNOT W22.01  ; Block Pointer Changed
+(400) W197 &1 W200  ; Block_Selected_Base, Current Programming Block ID
MOV(021) W198 DR0  ; Block Pointer Offset Calculated

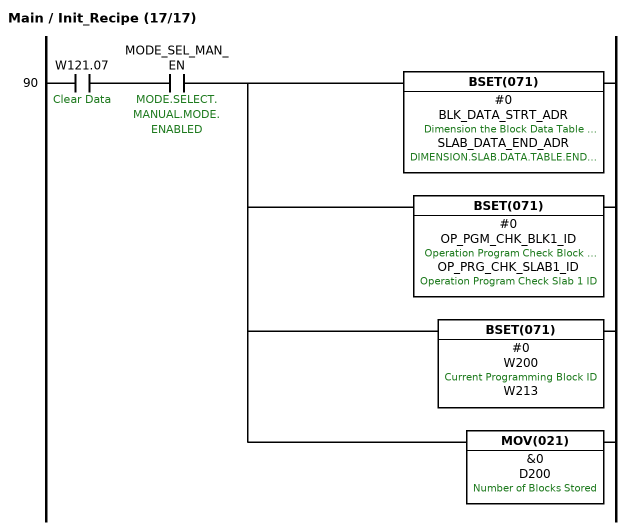
; rung 90
LD W121.07  ; Clear Data
AND MODE_SEL_MAN_EN  ; MODE.SELECT.MANUAL.MODE.ENABLED
BSET(071) #0 BLK_DATA_STRT_ADR SLAB_DATA_END_ADR  ; Dimension the Block Data Table - Start Address, DIMENSION.SLAB.DATA.TABLE.END.ADDRESS
BSET(071) #0 OP_PGM_CHK_BLK1_ID OP_PRG_CHK_SLAB1_ID  ; Operation Program Check Block 1 Block ID, Operation Program Check Slab 1 ID
BSET(071) #0 W200 W213  ; Current Programming Block ID
MOV(021) &0 D200  ; Number of Blocks Stored

### Section Init_Message_Display

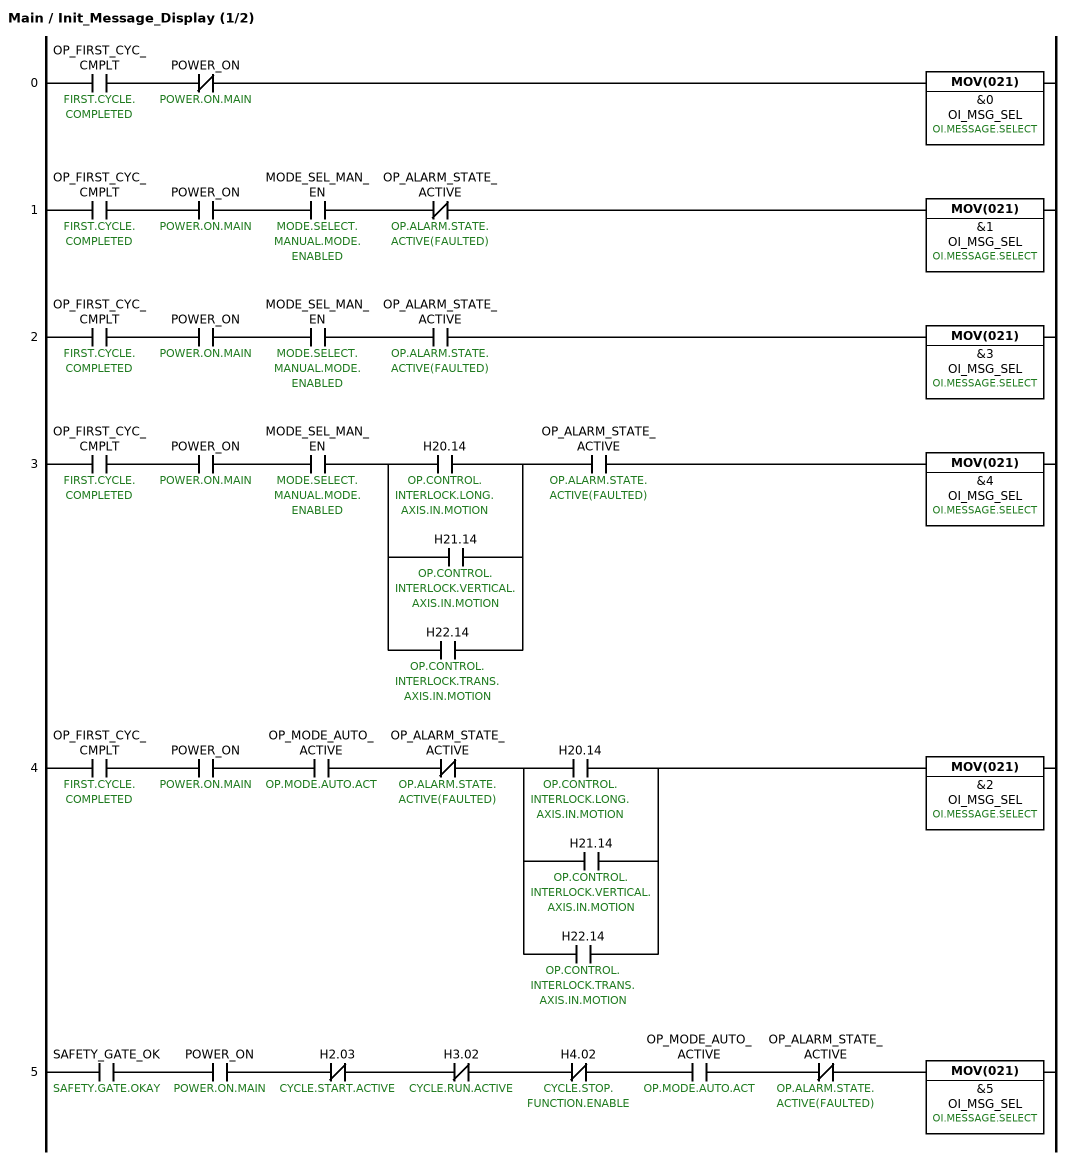
; rung 0
LD OP_FIRST_CYC_CMPLT  ; FIRST.CYCLE.COMPLETED
ANDNOT POWER_ON  ; POWER.ON.MAIN
MOV(021) &0 OI_MSG_SEL  ; OI.MESSAGE.SELECT
; rung 1
LD OP_FIRST_CYC_CMPLT  ; FIRST.CYCLE.COMPLETED
AND POWER_ON  ; POWER.ON.MAIN
AND MODE_SEL_MAN_EN  ; MODE.SELECT.MANUAL.MODE.ENABLED
ANDNOT OP_ALARM_STATE_ACTIVE  ; OP.ALARM.STATE.ACTIVE(FAULTED)
MOV(021) &1 OI_MSG_SEL  ; OI.MESSAGE.SELECT
; rung 2
LD OP_FIRST_CYC_CMPLT  ; FIRST.CYCLE.COMPLETED
AND POWER_ON  ; POWER.ON.MAIN
AND MODE_SEL_MAN_EN  ; MODE.SELECT.MANUAL.MODE.ENABLED
AND OP_ALARM_STATE_ACTIVE  ; OP.ALARM.STATE.ACTIVE(FAULTED)
MOV(021) &3 OI_MSG_SEL  ; OI.MESSAGE.SELECT
; rung 3
LD OP_FIRST_CYC_CMPLT  ; FIRST.CYCLE.COMPLETED
AND POWER_ON  ; POWER.ON.MAIN
AND MODE_SEL_MAN_EN  ; MODE.SELECT.MANUAL.MODE.ENABLED
LD H20.14  ; OP.CONTROL.INTERLOCK.LONG.AXIS.IN.MOTION
OR H21.14  ; OP.CONTROL.INTERLOCK.VERTICAL.AXIS.IN.MOTION
OR H22.14  ; OP.CONTROL.INTERLOCK.TRANS.AXIS.IN.MOTION
ANDLD
AND OP_ALARM_STATE_ACTIVE  ; OP.ALARM.STATE.ACTIVE(FAULTED)
MOV(021) &4 OI_MSG_SEL  ; OI.MESSAGE.SELECT
; rung 4
LD OP_FIRST_CYC_CMPLT  ; FIRST.CYCLE.COMPLETED
AND POWER_ON  ; POWER.ON.MAIN
AND OP_MODE_AUTO_ACTIVE  ; OP.MODE.AUTO.ACT
ANDNOT OP_ALARM_STATE_ACTIVE  ; OP.ALARM.STATE.ACTIVE(FAULTED)
LD H20.14  ; OP.CONTROL.INTERLOCK.LONG.AXIS.IN.MOTION
OR H21.14  ; OP.CONTROL.INTERLOCK.VERTICAL.AXIS.IN.MOTION
OR H22.14  ; OP.CONTROL.INTERLOCK.TRANS.AXIS.IN.MOTION
ANDLD
MOV(021) &2 OI_MSG_SEL  ; OI.MESSAGE.SELECT
; rung 5
LD SAFETY_GATE_OK  ; SAFETY.GATE.OKAY
AND POWER_ON  ; POWER.ON.MAIN
ANDNOT H2.03  ; CYCLE.START.ACTIVE
ANDNOT H3.02  ; CYCLE.RUN.ACTIVE
ANDNOT H4.02  ; CYCLE.STOP.FUNCTION.ENABLE
AND OP_MODE_AUTO_ACTIVE  ; OP.MODE.AUTO.ACT
ANDNOT OP_ALARM_STATE_ACTIVE  ; OP.ALARM.STATE.ACTIVE(FAULTED)
MOV(021) &5 OI_MSG_SEL  ; OI.MESSAGE.SELECT

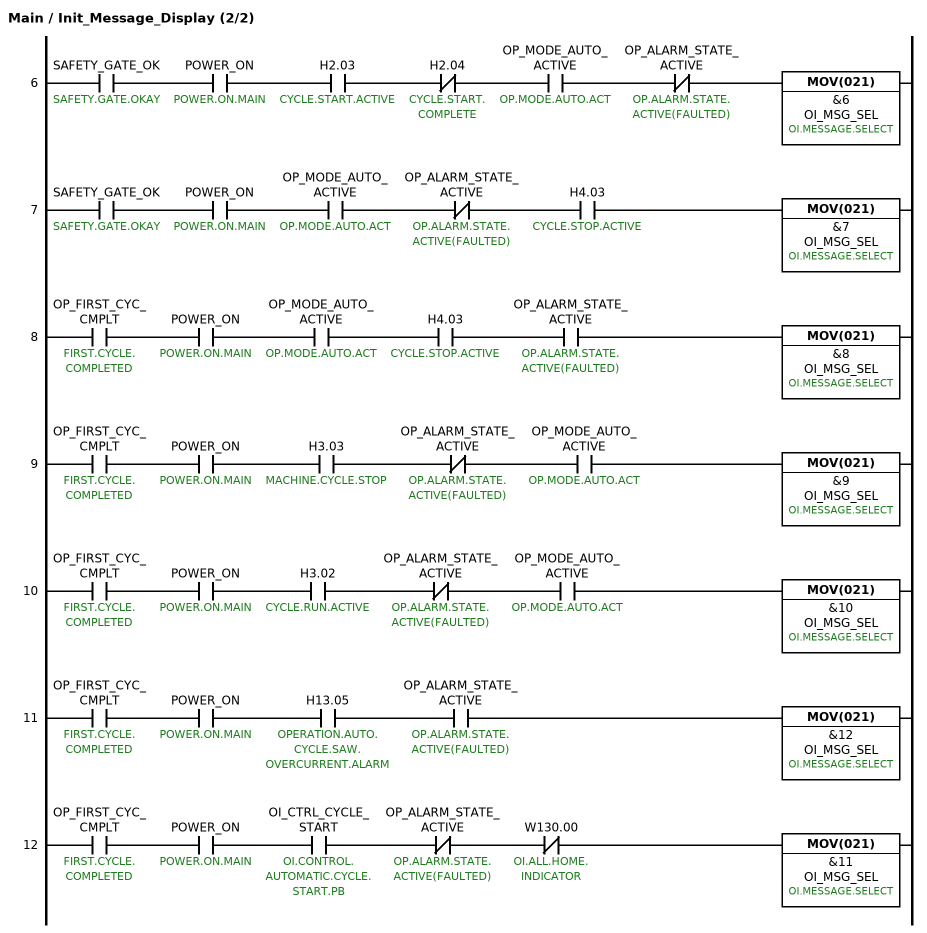
; rung 6
LD SAFETY_GATE_OK  ; SAFETY.GATE.OKAY
AND POWER_ON  ; POWER.ON.MAIN
AND H2.03  ; CYCLE.START.ACTIVE
ANDNOT H2.04  ; CYCLE.START.COMPLETE
AND OP_MODE_AUTO_ACTIVE  ; OP.MODE.AUTO.ACT
ANDNOT OP_ALARM_STATE_ACTIVE  ; OP.ALARM.STATE.ACTIVE(FAULTED)
MOV(021) &6 OI_MSG_SEL  ; OI.MESSAGE.SELECT
; rung 7
LD SAFETY_GATE_OK  ; SAFETY.GATE.OKAY
AND POWER_ON  ; POWER.ON.MAIN
AND OP_MODE_AUTO_ACTIVE  ; OP.MODE.AUTO.ACT
ANDNOT OP_ALARM_STATE_ACTIVE  ; OP.ALARM.STATE.ACTIVE(FAULTED)
AND H4.03  ; CYCLE.STOP.ACTIVE
MOV(021) &7 OI_MSG_SEL  ; OI.MESSAGE.SELECT
; rung 8
LD OP_FIRST_CYC_CMPLT  ; FIRST.CYCLE.COMPLETED
AND POWER_ON  ; POWER.ON.MAIN
AND OP_MODE_AUTO_ACTIVE  ; OP.MODE.AUTO.ACT
AND H4.03  ; CYCLE.STOP.ACTIVE
AND OP_ALARM_STATE_ACTIVE  ; OP.ALARM.STATE.ACTIVE(FAULTED)
MOV(021) &8 OI_MSG_SEL  ; OI.MESSAGE.SELECT
; rung 9
LD OP_FIRST_CYC_CMPLT  ; FIRST.CYCLE.COMPLETED
AND POWER_ON  ; POWER.ON.MAIN
AND H3.03  ; MACHINE.CYCLE.STOP
ANDNOT OP_ALARM_STATE_ACTIVE  ; OP.ALARM.STATE.ACTIVE(FAULTED)
AND OP_MODE_AUTO_ACTIVE  ; OP.MODE.AUTO.ACT
MOV(021) &9 OI_MSG_SEL  ; OI.MESSAGE.SELECT
; rung 10
LD OP_FIRST_CYC_CMPLT  ; FIRST.CYCLE.COMPLETED
AND POWER_ON  ; POWER.ON.MAIN
AND H3.02  ; CYCLE.RUN.ACTIVE
ANDNOT OP_ALARM_STATE_ACTIVE  ; OP.ALARM.STATE.ACTIVE(FAULTED)
AND OP_MODE_AUTO_ACTIVE  ; OP.MODE.AUTO.ACT
MOV(021) &10 OI_MSG_SEL  ; OI.MESSAGE.SELECT
; rung 11
LD OP_FIRST_CYC_CMPLT  ; FIRST.CYCLE.COMPLETED
AND POWER_ON  ; POWER.ON.MAIN
AND H13.05  ; OPERATION.AUTO.CYCLE.SAW.OVERCURRENT.ALARM
AND OP_ALARM_STATE_ACTIVE  ; OP.ALARM.STATE.ACTIVE(FAULTED)
MOV(021) &12 OI_MSG_SEL  ; OI.MESSAGE.SELECT
; rung 12
LD OP_FIRST_CYC_CMPLT  ; FIRST.CYCLE.COMPLETED
AND POWER_ON  ; POWER.ON.MAIN
AND OI_CTRL_CYCLE_START  ; OI.CONTROL.AUTOMATIC.CYCLE.START.PB
ANDNOT OP_ALARM_STATE_ACTIVE  ; OP.ALARM.STATE.ACTIVE(FAULTED)
ANDNOT W130.00  ; OI.ALL.HOME.INDICATOR
MOV(021) &11 OI_MSG_SEL  ; OI.MESSAGE.SELECT

### Section Init_Alarm_Display

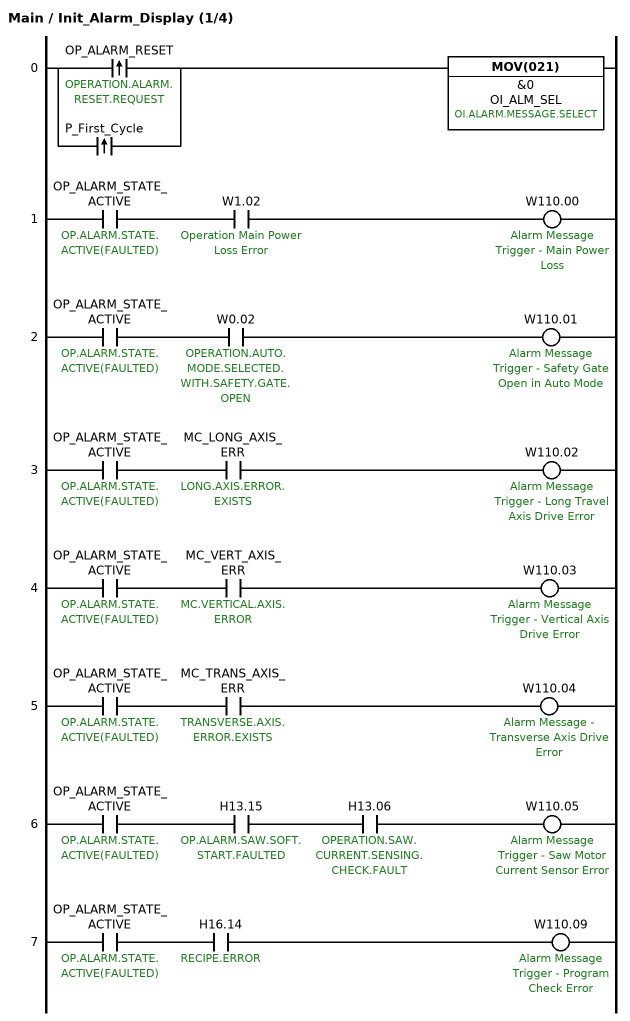
; rung 0
@LD OP_ALARM_RESET  ; OPERATION.ALARM.RESET.REQUEST
@OR P_First_Cycle
MOV(021) &0 OI_ALM_SEL  ; OI.ALARM.MESSAGE.SELECT
; rung 1
LD OP_ALARM_STATE_ACTIVE  ; OP.ALARM.STATE.ACTIVE(FAULTED)
AND W1.02  ; Operation Main Power Loss Error
OUT W110.00  ; Alarm Message Trigger - Main Power Loss
; rung 2
LD OP_ALARM_STATE_ACTIVE  ; OP.ALARM.STATE.ACTIVE(FAULTED)
AND W0.02  ; OPERATION.AUTO.MODE.SELECTED.WITH.SAFETY.GATE.OPEN
OUT W110.01  ; Alarm Message Trigger - Safety Gate Open in Auto Mode
; rung 3
LD OP_ALARM_STATE_ACTIVE  ; OP.ALARM.STATE.ACTIVE(FAULTED)
AND MC_LONG_AXIS_ERR  ; LONG.AXIS.ERROR.EXISTS
OUT W110.02  ; Alarm Message Trigger - Long Travel Axis Drive Error
; rung 4
LD OP_ALARM_STATE_ACTIVE  ; OP.ALARM.STATE.ACTIVE(FAULTED)
AND MC_VERT_AXIS_ERR  ; MC.VERTICAL.AXIS.ERROR
OUT W110.03  ; Alarm Message Trigger - Vertical Axis Drive Error
; rung 5
LD OP_ALARM_STATE_ACTIVE  ; OP.ALARM.STATE.ACTIVE(FAULTED)
AND MC_TRANS_AXIS_ERR  ; TRANSVERSE.AXIS.ERROR.EXISTS
OUT W110.04  ; Alarm Message - Transverse Axis Drive Error
; rung 6
LD OP_ALARM_STATE_ACTIVE  ; OP.ALARM.STATE.ACTIVE(FAULTED)
AND H13.15  ; OP.ALARM.SAW.SOFT.START.FAULTED
AND H13.06  ; OPERATION.SAW.CURRENT.SENSING.CHECK.FAULT
OUT W110.05  ; Alarm Message Trigger - Saw Motor Current Sensor Error
; rung 7
LD OP_ALARM_STATE_ACTIVE  ; OP.ALARM.STATE.ACTIVE(FAULTED)
AND H16.14  ; RECIPE.ERROR
OUT W110.09  ; Alarm Message Trigger - Program Check Error

